TYPE ST_Value :
STRUCT
	Setpoint	: REAL;
	Actual		: REAL;
END_STRUCT
END_TYPE

(* stored: Version 1.1.0.1, ProductVersion 3.1.4024.13
   DUT ST_Value: Id {beb28efd-48a5-0783-2b72-a8f209410c08} *)
